Staubli VAL3: recvTrajPtFull.pgx

public program recvTrajPtFull(bool& x_bFlag)
begin
  // receive message ID 14 data (prefix and header are in rosGenericMsg)
  rosTrajPtFMsg.prefix.nLength = rosGenericMsg.prefix.nLength
  rosTrajPtFMsg.header.nMsgType = rosGenericMsg.header.nMsgType
  rosTrajPtFMsg.header.nCommType = rosGenericMsg.header.nCommType
  rosTrajPtFMsg.header.nReplyCode = rosGenericMsg.header.nReplyCode

  call recvData(siTcpIpMotion, rosTrajPtFMsg.body.nData, nDataIn, x_bFlag)


//  // receive message ID 14 data (prefix and header are in rosGenericMsg)
//  l_nBytesRecv = 0
//  l_nIndex = 0
//
//  rosTrajPtFMsg.prefix.nLength = rosGenericMsg.prefix.nLength
//  rosTrajPtFMsg.header.nMsgType = rosGenericMsg.header.nMsgType
//  rosTrajPtFMsg.header.nCommType = rosGenericMsg.header.nCommType
//  rosTrajPtFMsg.header.nReplyCode = rosGenericMsg.header.nReplyCode
//
//  //while (l_nBytesRecv < (rosGenericMsg.prefix.nLength - 12))
//  while (l_nBytesRecv < 52)
//    l_nIndex = sioGet(siTcpIpMotion, l_nByte)
//    if (l_nIndex == -1)
//      if (l_nBytesRecv == 0)
//        // 11000: client is not connected?
//        if (nDataIn == 1)
//          nDataIn = -1
//        endIf
//      else
//        // 11000: connection lost
//        if (nDataIn == 1)
//          nDataIn = -1
//        endIf
//      endIf
//      bValidMsgBody = false
//      return
//    elseIf (l_nIndex == 1)
//      rosTrajPtFMsg.body.nData[l_nBytesRecv] = l_nByte
//      l_nBytesRecv = l_nBytesRecv + l_nIndex
//      nDataIn = 1
//    endIf
//  endWhile
//  bValidMsgBody = true
end
